PROGRAM Circuito_L3
VAR_INPUT
			Modo_Calibrar_L3 :BOOL;
END_VAR
VAR
		fbBomba_L3 :Equipo_Motor_ATV320;
		Totalizador_L3: Totalizador;//totalizador caudalimetro inferior
		Totalizador_L3_s: Totalizador;//totalizador caudalimetro superior
		Reset_TotL3:BOOL;
		Reset_TotL3_s: BOOL;
		PID_L3:FB_PID;
		ControlValv_ioLink_V1:ControlValv_ioLink;
		ControlValv_ioLink_V2: ControlValv_ioLink;
		ControlValv_ioLink_V3: ControlValv_ioLink;
		ControlValv_ioLink_V4: ControlValv_ioLink;
		Falla_L3_V1:BOOL;
		Falla_L3_V2:BOOL;
		Falla_L3_V3:BOOL;
		Falla_L3_V4:BOOL;
		Balanza_PU1_WT3: Balanza;
		TOF_calibradoIBC: TOF;
		
		auxHS:BOOL;
		dHS:DINT;
		PID_L3_SP:REAL;
		PID_L3_auto:BOOL;
		PID_L3_reset:BOOL;
		PID_L3_manual:REAL;
		PID_L3_bMuerta:REAL := 5;
		PID_L3_Kp:REAL := 0.1;
		PID_L3_Ti:REAL := 100;
		PID_L3_PV:REAL;
		Dosis_L3	:REAL;
		TiempoInyeccion_L3	:DINT;
		Peso	:REAL;
		Offset_L3:REAL;
		Inyeccion_L3:BOOL;

		Volumen_L3:Real;
	Calculo_caudal_L3: Calculo_caudal;
	CorrecionCaudalxOffset_L3: CorrecionCaudalxOffset;
	tInyeccion: TON;
	Total :REAL;
	Totalant	:REAL;
	auxIniCal:BOOL;
	AuxVol:REAL;
	CA1_L3_V1_CmdA_Man :BOOL;
	CA1_L3_V4_CmdA_Man :BOOL;
	TDemoraInyectar: TON;
	SetDemoraInyeccion: REAL;
	TiempoDeInyeccion:TIME;
	Tiempo_TIME_to_seg_InyCal: Tiempo_TIME_to_seg;
	AuxInyCal:TIME;
	Tiempo_seg_to_TIME_DemoraInyec: Tiempo_seg_to_TIME;
	AuxTDemoraInyec: TIME;
	IniTotalFT2:REAL;
	Auxconsumo:REAL;
	ProductoAsociado: STRING;
	Lavagem_Circuito03: Lavagem;
	Filtro2_Teste: Filtro2;
	PID_GENERICO_0: PID_GENERICO;
END_VAR
VAR PERSISTENT
	UltimaCalibracao	:UDINT;	//Data e hora da ultima calibração
END_VAR
VAR // added by the converter: edge detectors and wires of the graphical bodies
    _w1, _w2, _w3, _w4, _w5, _w6, _w7, _w8, _w9, _w10, _w11, _w12, _w13 : BOOL;
    _ft1 : F_TRIG;
    _rt1, _rt2 : R_TRIG;
END_VAR

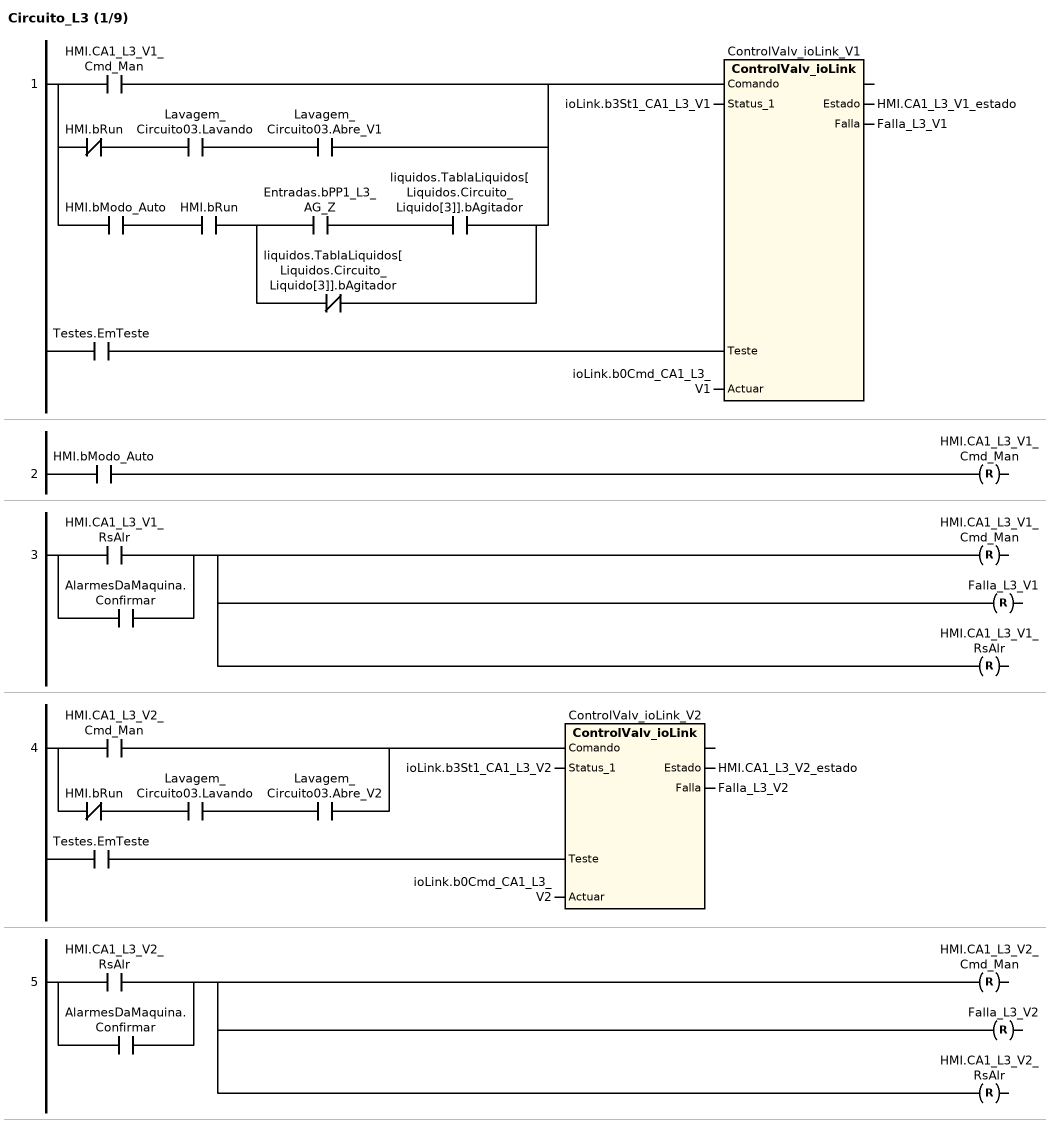
// NETWORK 1
ControlValv_ioLink_V1(
    Comando := HMI.CA1_L3_V1_Cmd_Man OR NOT HMI.bRun AND Lavagem_Circuito03.Lavando AND Lavagem_Circuito03.Abre_V1 OR HMI.bModo_Auto AND HMI.bRun AND (Entradas.bPP1_L3_AG_Z AND (liquidos.TablaLiquidos[Liquidos.Circuito_Liquido[3]].bAgitador) OR NOT (liquidos.TablaLiquidos[Liquidos.Circuito_Liquido[3]].bAgitador)),
    Status_1 := ioLink.b3St1_CA1_L3_V1,
    Teste := Testes.EmTeste,
    Actuar := ioLink.b0Cmd_CA1_L3_V1,
    Estado => HMI.CA1_L3_V1_estado,
    Falla => Falla_L3_V1); // ControlValv_ioLink

// NETWORK 2
HMI.CA1_L3_V1_Cmd_Man R= HMI.bModo_Auto;

// NETWORK 3
_w1 := HMI.CA1_L3_V1_RsAlr OR AlarmesDaMaquina.Confirmar;
HMI.CA1_L3_V1_Cmd_Man R= _w1;
Falla_L3_V1 R= _w1;
HMI.CA1_L3_V1_RsAlr R= _w1;

// NETWORK 4
ControlValv_ioLink_V2(
    Comando := HMI.CA1_L3_V2_Cmd_Man OR NOT HMI.bRun AND Lavagem_Circuito03.Lavando AND Lavagem_Circuito03.Abre_V2,
    Status_1 := ioLink.b3St1_CA1_L3_V2,
    Teste := Testes.EmTeste,
    Actuar := ioLink.b0Cmd_CA1_L3_V2,
    Estado => HMI.CA1_L3_V2_estado,
    Falla => Falla_L3_V2); // ControlValv_ioLink

// NETWORK 5
_w2 := HMI.CA1_L3_V2_RsAlr OR AlarmesDaMaquina.Confirmar;
HMI.CA1_L3_V2_Cmd_Man R= _w2;
Falla_L3_V2 R= _w2;
HMI.CA1_L3_V2_RsAlr R= _w2;

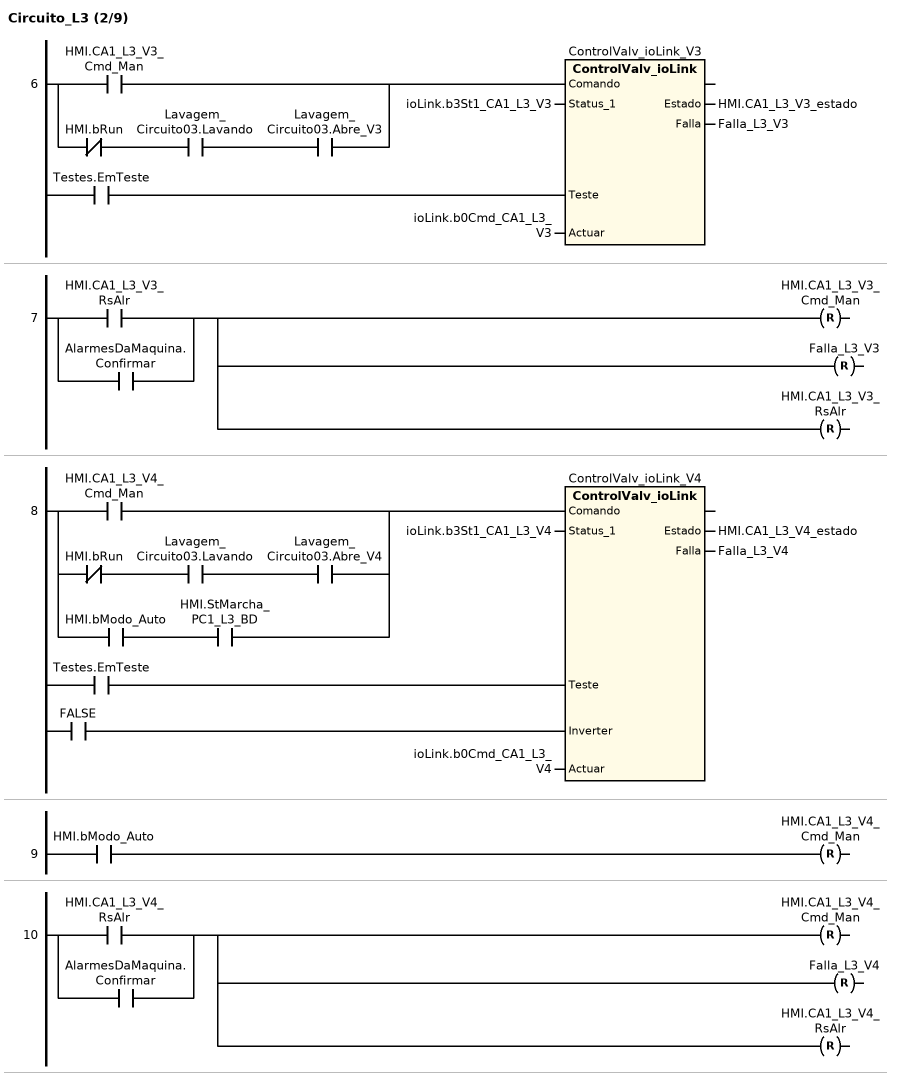
// NETWORK 6
ControlValv_ioLink_V3(
    Comando := HMI.CA1_L3_V3_Cmd_Man OR NOT HMI.bRun AND Lavagem_Circuito03.Lavando AND Lavagem_Circuito03.Abre_V3,
    Status_1 := ioLink.b3St1_CA1_L3_V3,
    Teste := Testes.EmTeste,
    Actuar := ioLink.b0Cmd_CA1_L3_V3,
    Estado => HMI.CA1_L3_V3_estado,
    Falla => Falla_L3_V3); // ControlValv_ioLink

// NETWORK 7
_w3 := HMI.CA1_L3_V3_RsAlr OR AlarmesDaMaquina.Confirmar;
HMI.CA1_L3_V3_Cmd_Man R= _w3;
Falla_L3_V3 R= _w3;
HMI.CA1_L3_V3_RsAlr R= _w3;

// NETWORK 8
ControlValv_ioLink_V4(
    Comando := HMI.CA1_L3_V4_Cmd_Man OR NOT HMI.bRun AND Lavagem_Circuito03.Lavando AND Lavagem_Circuito03.Abre_V4 OR HMI.bModo_Auto AND HMI.StMarcha_PC1_L3_BD,
    Status_1 := ioLink.b3St1_CA1_L3_V4,
    Teste := Testes.EmTeste,
    Inverter := FALSE,
    Actuar := ioLink.b0Cmd_CA1_L3_V4,
    Estado => HMI.CA1_L3_V4_estado,
    Falla => Falla_L3_V4); // ControlValv_ioLink

// NETWORK 9
HMI.CA1_L3_V4_Cmd_Man R= HMI.bModo_Auto;

// NETWORK 10
_w4 := HMI.CA1_L3_V4_RsAlr OR AlarmesDaMaquina.Confirmar;
HMI.CA1_L3_V4_Cmd_Man R= _w4;
Falla_L3_V4 R= _w4;
HMI.CA1_L3_V4_RsAlr R= _w4;

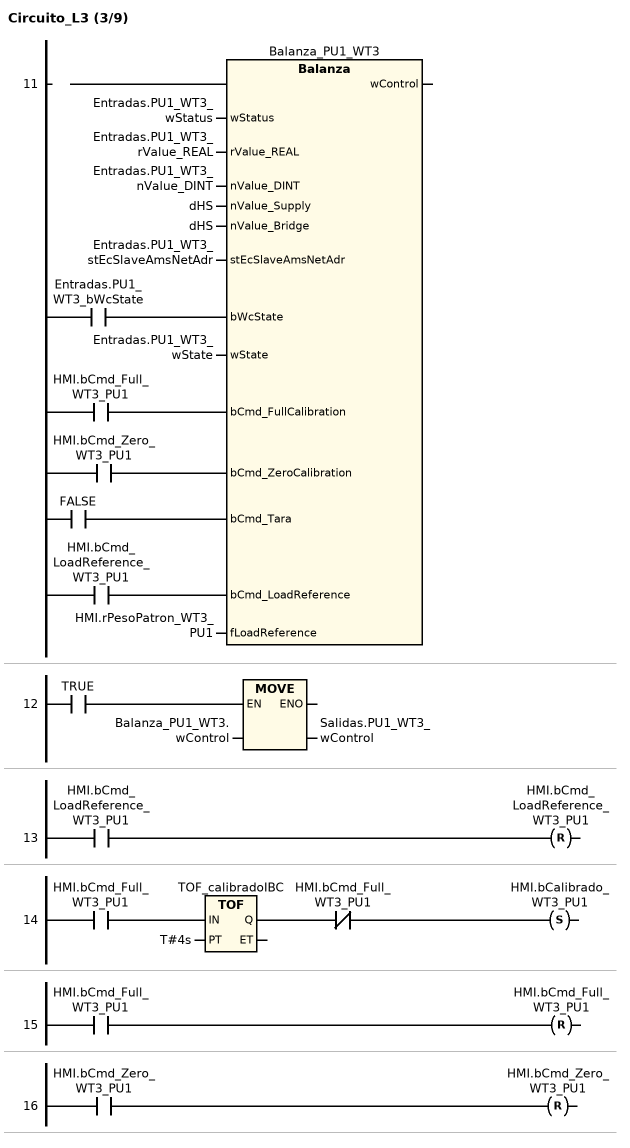
// NETWORK 11
Balanza_PU1_WT3(
    wStatus := Entradas.PU1_WT3_wStatus,
    rValue_REAL := Entradas.PU1_WT3_rValue_REAL,
    nValue_DINT := Entradas.PU1_WT3_nValue_DINT,
    nValue_Supply := dHS,
    nValue_Bridge := dHS,
    stEcSlaveAmsNetAdr := Entradas.PU1_WT3_stEcSlaveAmsNetAdr,
    bWcState := Entradas.PU1_WT3_bWcState,
    wState := Entradas.PU1_WT3_wState,
    bCmd_FullCalibration := HMI.bCmd_Full_WT3_PU1,
    bCmd_ZeroCalibration := HMI.bCmd_Zero_WT3_PU1,
    bCmd_Tara := FALSE,
    bCmd_LoadReference := HMI.bCmd_LoadReference_WT3_PU1,
    fLoadReference := HMI.rPesoPatron_WT3_PU1); // Balanza

// NETWORK 12
Salidas.PU1_WT3_wControl := Balanza_PU1_WT3.wControl;

// NETWORK 13
HMI.bCmd_LoadReference_WT3_PU1 R= HMI.bCmd_LoadReference_WT3_PU1;

// NETWORK 14
TOF_calibradoIBC(IN := HMI.bCmd_Full_WT3_PU1, PT := T#4s); // TOF
HMI.bCalibrado_WT3_PU1 S= TOF_calibradoIBC.Q AND NOT HMI.bCmd_Full_WT3_PU1;

// NETWORK 15
HMI.bCmd_Full_WT3_PU1 R= HMI.bCmd_Full_WT3_PU1;

// NETWORK 16
HMI.bCmd_Zero_WT3_PU1 R= HMI.bCmd_Zero_WT3_PU1;

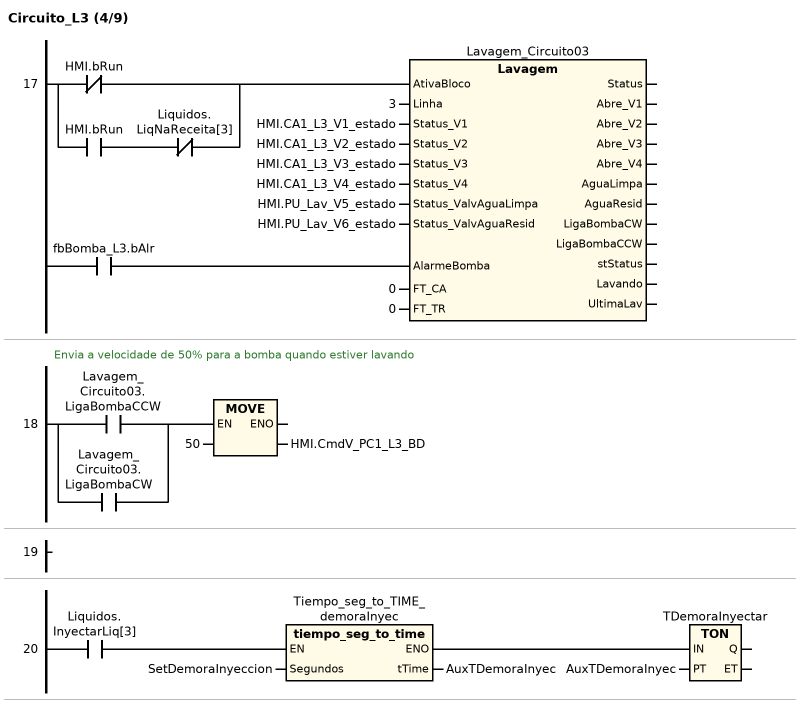
// NETWORK 17
Lavagem_Circuito03(
    AtivaBloco := NOT HMI.bRun OR HMI.bRun AND NOT Liquidos.LiqNaReceita[3],
    Linha := 3,
    Status_V1 := HMI.CA1_L3_V1_estado,
    Status_V2 := HMI.CA1_L3_V2_estado,
    Status_V3 := HMI.CA1_L3_V3_estado,
    Status_V4 := HMI.CA1_L3_V4_estado,
    Status_ValvAguaLimpa := HMI.PU_Lav_V5_estado,
    Status_ValvAguaResid := HMI.PU_Lav_V6_estado,
    AlarmeBomba := fbBomba_L3.bAlr,
    FT_CA := 0,
    FT_TR := 0); // Lavagem

// NETWORK 18
// Envia a velocidade de 50% para a bomba quando estiver lavando
IF Lavagem_Circuito03.LigaBombaCCW OR Lavagem_Circuito03.LigaBombaCW THEN HMI.CmdV_PC1_L3_BD := 50; END_IF

// NETWORK 19

// NETWORK 20
_w5 := Liquidos.InyectarLiq[3];
IF _w5 THEN
    Tiempo_seg_to_TIME_demoraInyec(Segundos := SetDemoraInyeccion, tTime => AuxTDemoraInyec); // tiempo_seg_to_time
END_IF
TDemoraInyectar(IN := _w5, PT := AuxTDemoraInyec); // TON

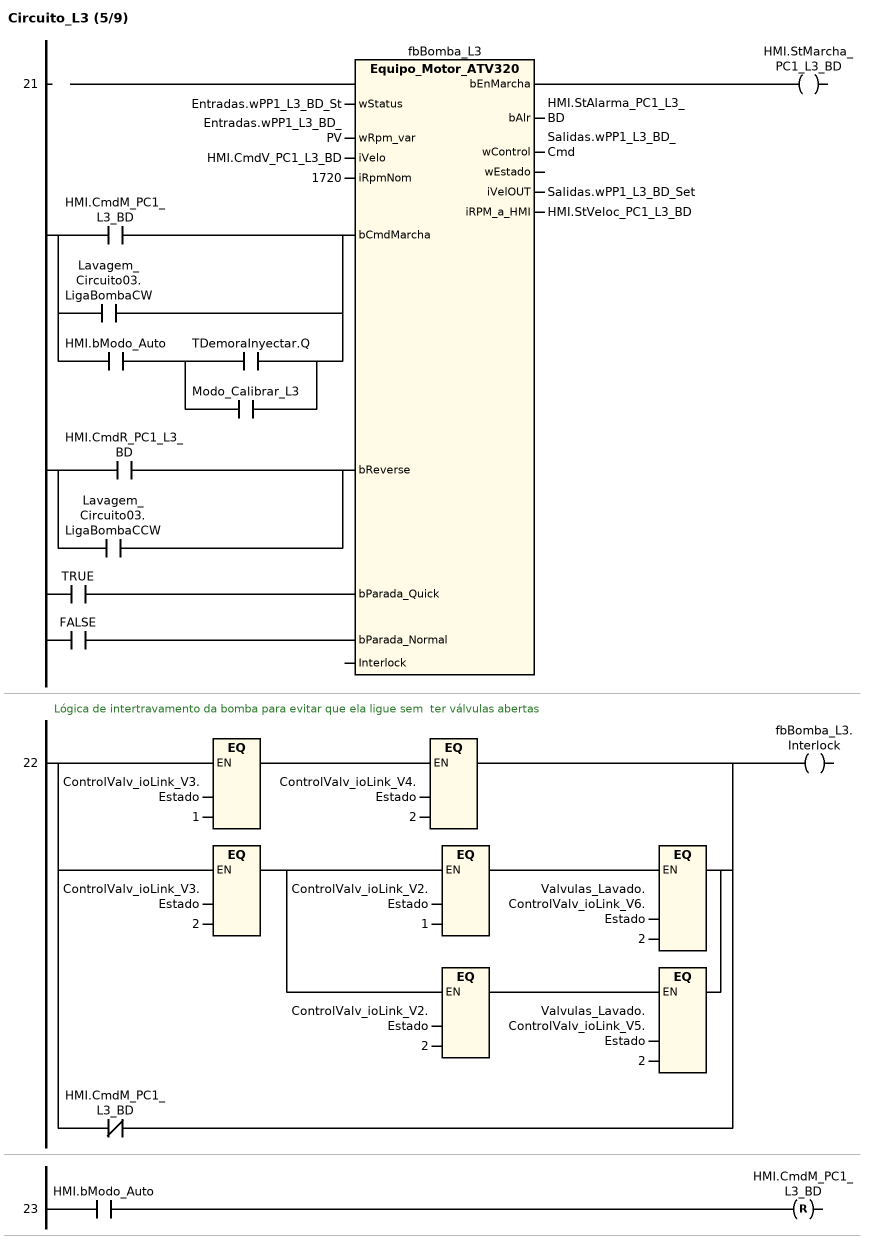
// NETWORK 21
fbBomba_L3(
    wStatus := Entradas.wPP1_L3_BD_St,
    wRpm_var := Entradas.wPP1_L3_BD_PV,
    iVelo := HMI.CmdV_PC1_L3_BD,
    iRpmNom := 1720,
    bCmdMarcha := HMI.CmdM_PC1_L3_BD OR Lavagem_Circuito03.LigaBombaCW OR HMI.bModo_Auto AND (TDemoraInyectar.Q OR Modo_Calibrar_L3),
    bReverse := HMI.CmdR_PC1_L3_BD OR Lavagem_Circuito03.LigaBombaCCW,
    bParada_Quick := TRUE,
    bParada_Normal := FALSE,
    bAlr => HMI.StAlarma_PC1_L3_BD,
    wControl => Salidas.wPP1_L3_BD_Cmd,
    iVelOUT => Salidas.wPP1_L3_BD_Set,
    iRPM_a_HMI => HMI.StVeloc_PC1_L3_BD); // Equipo_Motor_ATV320
HMI.StMarcha_PC1_L3_BD := fbBomba_L3.bEnMarcha;

// NETWORK 22
// Lógica de intertravamento da bomba para evitar que ela ligue sem  ter válvulas abertas
_w6 := NOT HMI.CmdM_PC1_L3_BD;
IF NOT _w6 THEN
    _w7 := ControlValv_ioLink_V3.Estado = 2;
    _w6 := ControlValv_ioLink_V3.Estado = 1 AND ControlValv_ioLink_V4.Estado = 2 OR (_w7 AND ControlValv_ioLink_V2.Estado = 1 AND Valvulas_Lavado.ControlValv_ioLink_V6.Estado = 2 OR _w7 AND ControlValv_ioLink_V2.Estado = 2 AND Valvulas_Lavado.ControlValv_ioLink_V5.Estado = 2);
END_IF
fbBomba_L3.Interlock := _w6;

// NETWORK 23
HMI.CmdM_PC1_L3_BD R= HMI.bModo_Auto;

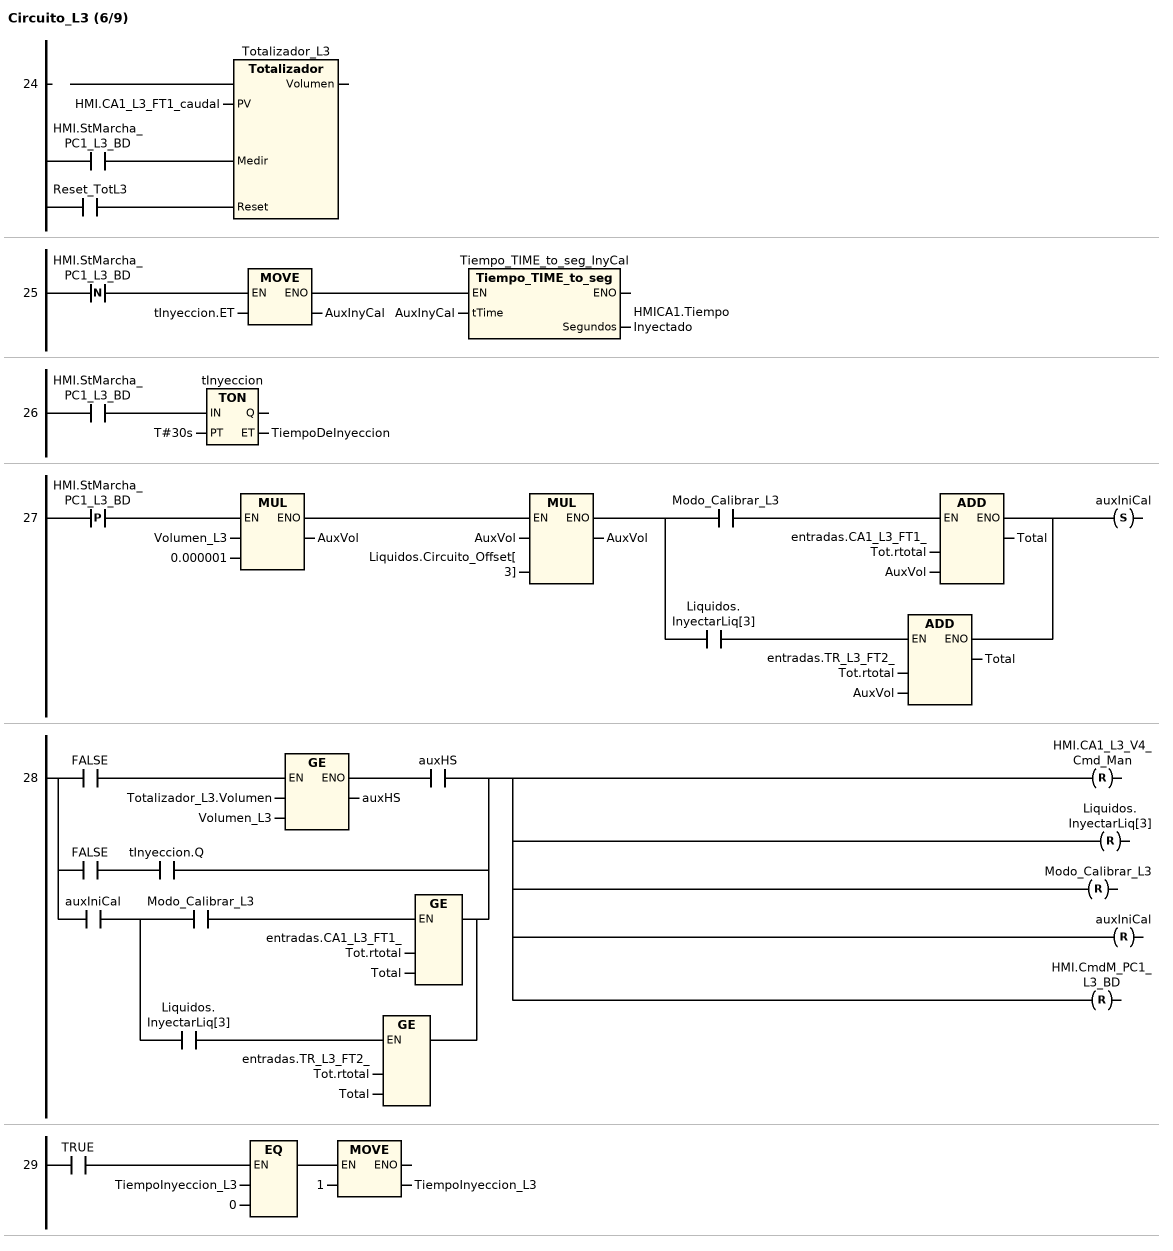
// NETWORK 24
Totalizador_L3(PV := HMI.CA1_L3_FT1_caudal, Medir := HMI.StMarcha_PC1_L3_BD, Reset := Reset_TotL3); // Totalizador

// NETWORK 25
_ft1(CLK := HMI.StMarcha_PC1_L3_BD);
_w8 := _ft1.Q;
IF _w8 THEN AuxInyCal := tInyeccion.ET; END_IF
IF _w8 THEN
    Tiempo_TIME_to_seg_InyCal(tTime := AuxInyCal, Segundos => HMICA1.TiempoInyectado); // Tiempo_TIME_to_seg
END_IF

// NETWORK 26
tInyeccion(IN := HMI.StMarcha_PC1_L3_BD, PT := T#30s, ET => TiempoDeInyeccion); // TON

// NETWORK 27
_rt1(CLK := HMI.StMarcha_PC1_L3_BD);
_w9 := _rt1.Q;
IF _w9 THEN AuxVol := Volumen_L3 * 0.000001; END_IF
IF _w9 THEN AuxVol := AuxVol * Liquidos.Circuito_Offset[3]; END_IF
IF _w9 AND Modo_Calibrar_L3 THEN Total := entradas.CA1_L3_FT1_Tot.rtotal + AuxVol; END_IF
IF _w9 AND Liquidos.InyectarLiq[3] THEN Total := entradas.TR_L3_FT2_Tot.rtotal + AuxVol; END_IF
auxIniCal S= _w9 AND Modo_Calibrar_L3 OR _w9 AND Liquidos.InyectarLiq[3];

// NETWORK 28
IF FALSE THEN auxHS := Totalizador_L3.Volumen >= Volumen_L3; END_IF
_w10 := FALSE AND auxHS OR FALSE AND tInyeccion.Q OR (auxIniCal AND Modo_Calibrar_L3 AND entradas.CA1_L3_FT1_Tot.rtotal >= Total OR auxIniCal AND Liquidos.InyectarLiq[3] AND entradas.TR_L3_FT2_Tot.rtotal >= Total);
HMI.CA1_L3_V4_Cmd_Man R= _w10;
Liquidos.InyectarLiq[3] R= _w10;
Modo_Calibrar_L3 R= _w10;
auxIniCal R= _w10;
HMI.CmdM_PC1_L3_BD R= _w10;

// NETWORK 29
IF TiempoInyeccion_L3 = 0 THEN TiempoInyeccion_L3 := 1; END_IF

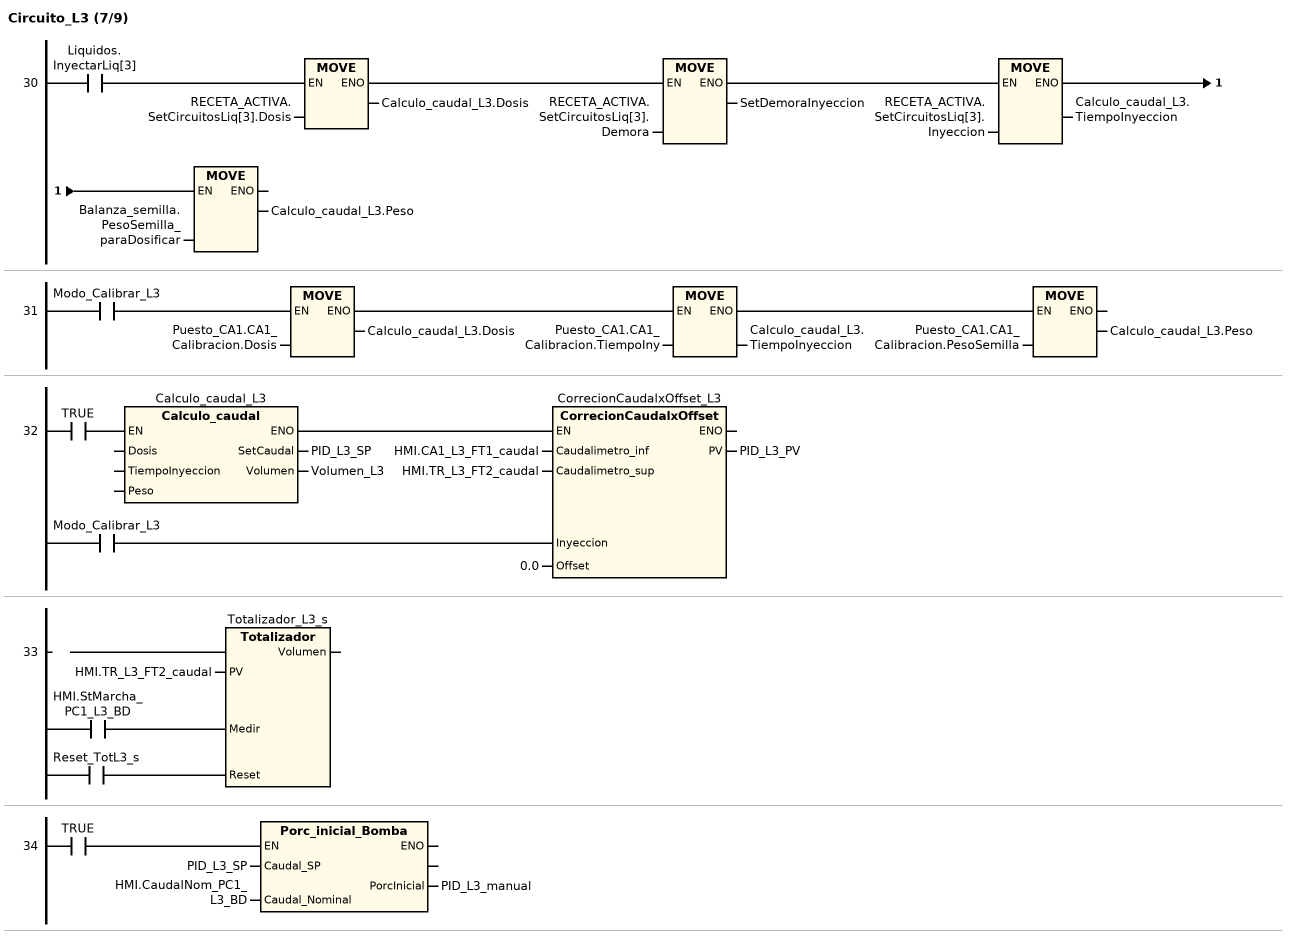
// NETWORK 30
_w11 := Liquidos.InyectarLiq[3];
IF _w11 THEN Calculo_caudal_L3.Dosis := RECETA_ACTIVA.SetCircuitosLiq[3].Dosis; END_IF
IF _w11 THEN SetDemoraInyeccion := RECETA_ACTIVA.SetCircuitosLiq[3].Demora; END_IF
IF _w11 THEN Calculo_caudal_L3.TiempoInyeccion := RECETA_ACTIVA.SetCircuitosLiq[3].Inyeccion; END_IF
IF _w11 THEN Calculo_caudal_L3.Peso := Balanza_semilla.PesoSemilla_paraDosificar; END_IF

// NETWORK 31
_w12 := Modo_Calibrar_L3;
IF _w12 THEN Calculo_caudal_L3.Dosis := Puesto_CA1.CA1_Calibracion.Dosis; END_IF
IF _w12 THEN Calculo_caudal_L3.TiempoInyeccion := Puesto_CA1.CA1_Calibracion.TiempoIny; END_IF
IF _w12 THEN Calculo_caudal_L3.Peso := Puesto_CA1.CA1_Calibracion.PesoSemilla; END_IF

// NETWORK 32
Calculo_caudal_L3(SetCaudal => PID_L3_SP, Volumen => Volumen_L3); // Calculo_caudal
CorrecionCaudalxOffset_L3(
    Caudalimetro_inf := HMI.CA1_L3_FT1_caudal,
    Caudalimetro_sup := HMI.TR_L3_FT2_caudal,
    Inyeccion := Modo_Calibrar_L3,
    Offset := 0.0,
    PV => PID_L3_PV); // CorrecionCaudalxOffset

// NETWORK 33
Totalizador_L3_s(PV := HMI.TR_L3_FT2_caudal, Medir := HMI.StMarcha_PC1_L3_BD, Reset := Reset_TotL3_s); // Totalizador

// NETWORK 34
Porc_inicial_Bomba(Caudal_SP := PID_L3_SP, Caudal_Nominal := HMI.CaudalNom_PC1_L3_BD, PorcInicial => PID_L3_manual);

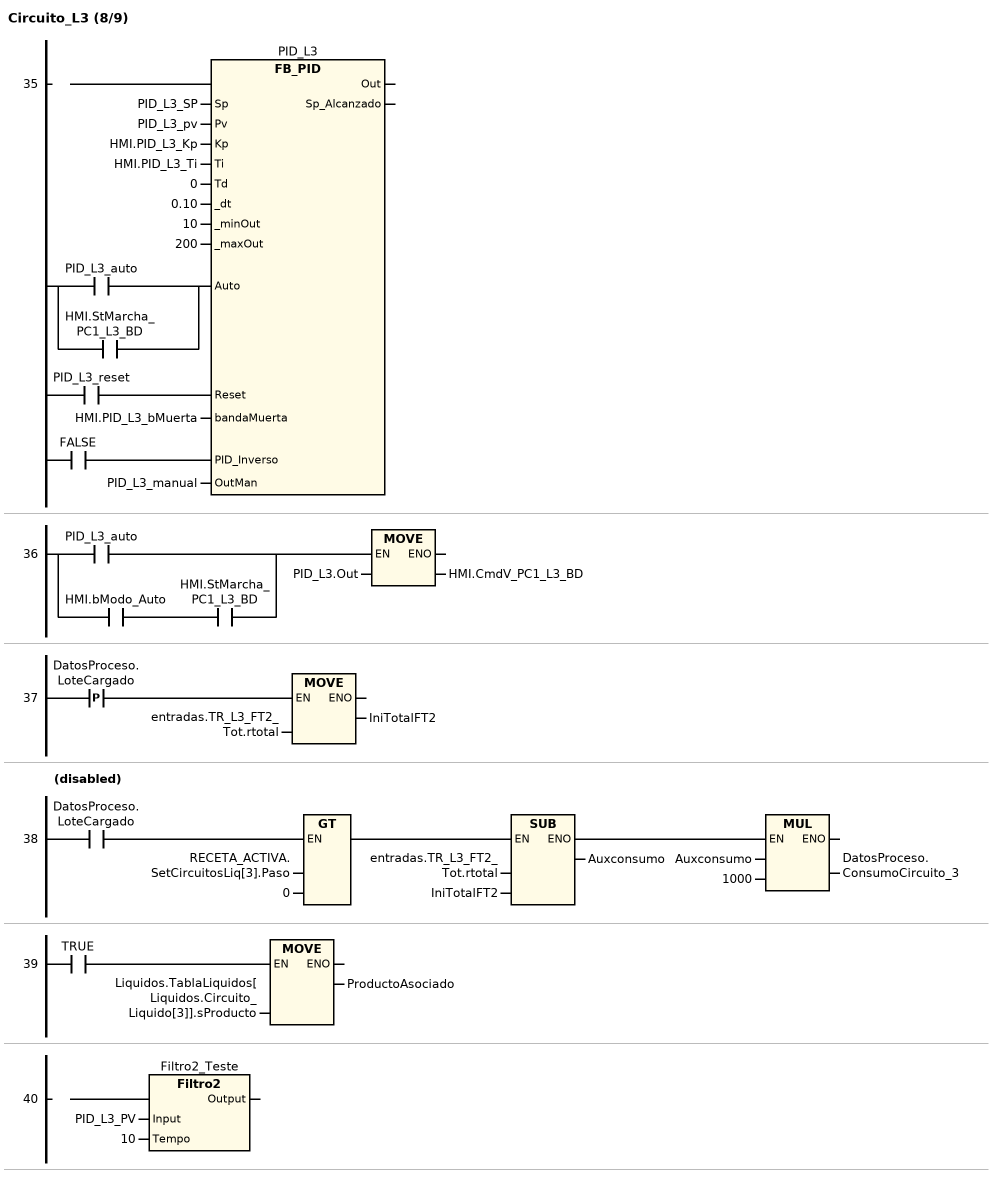
// NETWORK 35
PID_L3(
    Sp := PID_L3_SP,
    Pv := PID_L3_pv,
    Kp := HMI.PID_L3_Kp,
    Ti := HMI.PID_L3_Ti,
    Td := 0,
    _dt := 0.10,
    _minOut := 10,
    _maxOut := 200,
    Auto := PID_L3_auto OR HMI.StMarcha_PC1_L3_BD,
    Reset := PID_L3_reset,
    bandaMuerta := HMI.PID_L3_bMuerta,
    PID_Inverso := FALSE,
    OutMan := PID_L3_manual); // FB_PID

// NETWORK 36
IF PID_L3_auto OR HMI.bModo_Auto AND HMI.StMarcha_PC1_L3_BD THEN HMI.CmdV_PC1_L3_BD := PID_L3.Out; END_IF

// NETWORK 37
_rt2(CLK := DatosProceso.LoteCargado);
IF _rt2.Q THEN IniTotalFT2 := entradas.TR_L3_FT2_Tot.rtotal; END_IF

// NETWORK 38 (disabled)
// _w13 := DatosProceso.LoteCargado AND RECETA_ACTIVA.SetCircuitosLiq[3].Paso > 0;
// IF _w13 THEN Auxconsumo := entradas.TR_L3_FT2_Tot.rtotal - IniTotalFT2; END_IF
// IF _w13 THEN DatosProceso.ConsumoCircuito_3 := Auxconsumo * 1000; END_IF

// NETWORK 39
ProductoAsociado := Liquidos.TablaLiquidos[Liquidos.Circuito_Liquido[3]].sProducto;

// NETWORK 40
Filtro2_Teste(Input := PID_L3_PV, Tempo := 10); // Filtro2

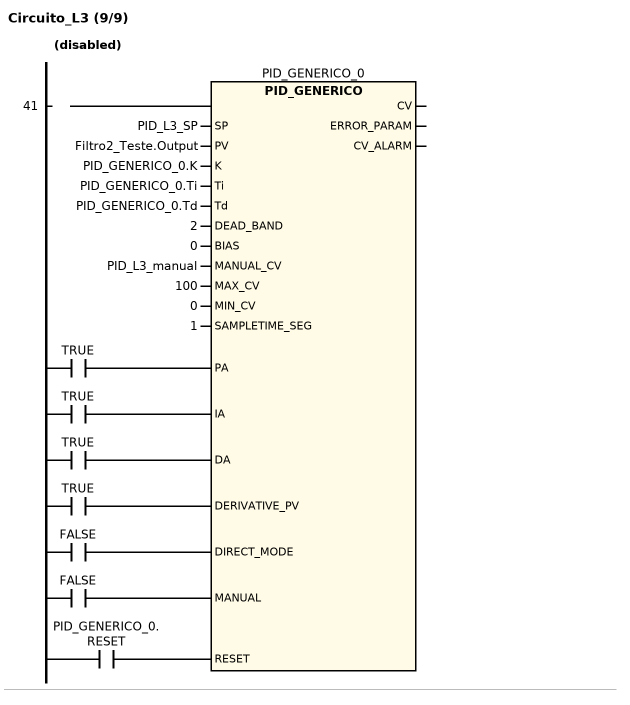
// NETWORK 41 (disabled)
// PID_GENERICO_0(
//     SP := PID_L3_SP,
//     PV := Filtro2_Teste.Output,
//     K := PID_GENERICO_0.K,
//     Ti := PID_GENERICO_0.Ti,
//     Td := PID_GENERICO_0.Td,
//     DEAD_BAND := 2,
//     BIAS := 0,
//     MANUAL_CV := PID_L3_manual,
//     MAX_CV := 100,
//     MIN_CV := 0,
//     SAMPLETIME_SEG := 1,
//     PA := TRUE,
//     IA := TRUE,
//     DA := TRUE,
//     DERIVATIVE_PV := TRUE,
//     DIRECT_MODE := FALSE,
//     MANUAL := FALSE,
//     RESET := PID_GENERICO_0.RESET); // PID_GENERICO

END_PROGRAM

(* stored: Version 1.1.0.1, ProductVersion 3.1.4024.14
   POU Circuito_L3: Id {096ad54d-021d-450a-af48-68159ba5a115}, SpecialFunc None *)
